Fanuc KAREL source: NC0002.KL

-- PROVISIONAL review KL for V940-1; original PC SHA256 93a371964678f7e18c0097c2017e2fdbbb75196df4860795077361318d1c93b4
-- Incomplete behavior may be omitted. Consult companion uncertainty JSON. Do not deploy.
PROGRAM NC0002
%NOLOCKGROUP
-- UNRESOLVED_LOCAL_POOL 1 cells at code offset 3; source declarations unknown
-- DIRECT_LOCAL_WORD_ACCESS alone does not prove INTEGER, REAL, or BOOLEAN
BEGIN
  -- V9_EXPOSED_INDEXED_TABLE_HINT layout=0001; 2 counted words exposed once; source arms/runtime held
  -- V9_CONDITION_STACK_HINT 1 bounded expression windows; static native code-base-relative target link; source arms held
  -- V9_BRANCH_PAIR_HINT routine=R 79->+67 7A->+95
  -- UNRESOLVED_PC offsets 0-8; opcodes 2B,2C,7B
  -- UNRESOLVED_PC offsets 13-20; opcodes 9D,23
  -- UNRESOLVED_PC offsets 25-38; opcodes 21,9D,57,79
  -- UNRESOLVED_PC offsets 43-57; opcodes 21,9D,52,23
  -- UNRESOLVED_PC offsets 62-67; opcodes 7A
  -- UNRESOLVED_PC offsets 72-90; opcodes 21,2E,52,23
  -- UNRESOLVED_PC offsets 100-104; opcodes 7F
  -- UNRESOLVED_PC offsets 109-113; opcodes 27,AA
  -- UNRESOLVED_PC offsets 118-122; opcodes 7F
END NC0002
